// TIA Portal project "Project400 pid control implementation" (V20)

(* hardware
DEVICE "HMI_1"  KTP400 Basic PN
   slot 0: "HMI_1"  KTP400 Basic PN  6AV2 123-2DB03-0AX0  17.0.0.0
   slot 1: "HMI_RT_1"  KTP400 Basic PN  6AV2 123-2DB03-0AX0  17.0.0.0
   slot 5: "HMI_1.IE_CP_1"  PROFINET Interface  17.0.0.0
      slot 1: "PROFINET Interface_1"  PROFINET Interface
         slot 1: "Port_1"  Port
DEVICE "S7-1200 station_1"  S7-1200 Station
   slot 0: "Rack_0"  S7-1200 Rack  Rack  V1.0
   slot 1: "PLC_1"  CPU 1215C AC/DC/Rly  6ES7 215-1BG31-0XB0  V3.0
*)

// ===== PLC "PLC_1"  CPU 1215C AC/DC/Rly =====

VAR_GLOBAL   // PLC tag table "Default tag table"
   "Temperature_SP" AT %MD0 : Real;
   "Temperature_RV" AT %MD4 : Real;
   "Manual_output" AT %MD8 : Real;
   "Manual_mode" AT %M12.0 : Bool;
   "Scale_output" AT %MW14 : Word;
   "PID_on" AT %Q0.0 : Bool;
   "Man_pb" AT %M12.1 : Bool;
   "auto_pb" AT %M12.2 : Bool;
END_VAR

ORGANIZATION_BLOCK "Main"   // OB1, LAD, ProgramCycle
TITLE = "Main Program Sweep (Cycle)"
{ S7_Optimized_Access := 'TRUE' }
VERSION : 0.1
BEGIN

REGION Network 1: Auto/manual Controller
END_REGION

REGION Network 3
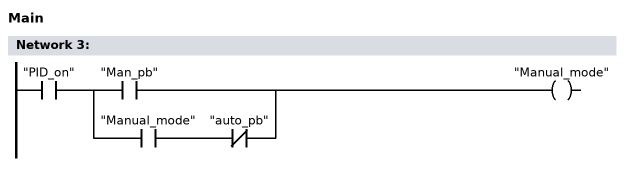
   RUNG wire#powerrail
      Contact( "PID_on" )
      wire#w1
      Contact( "Man_pb" )
      wire#w2
      Coil( "Manual_mode" )
   END_RUNG
   RUNG wire#w1
      Contact( "Manual_mode" )
      I_Contact( "auto_pb" )
   END_RUNG wire#w2
   // the same network as SCL:
   "Manual_mode" := "PID_on" AND ("Man_pb" OR ("Manual_mode" AND NOT "auto_pb"));
END_REGION
END_ORGANIZATION_BLOCK

ORGANIZATION_BLOCK "PID_CONTROLLER"   // OB30, LAD, CyclicInterrupt
{ S7_Optimized_Access := 'TRUE' }
VERSION : 0.1
BEGIN

REGION Network 1
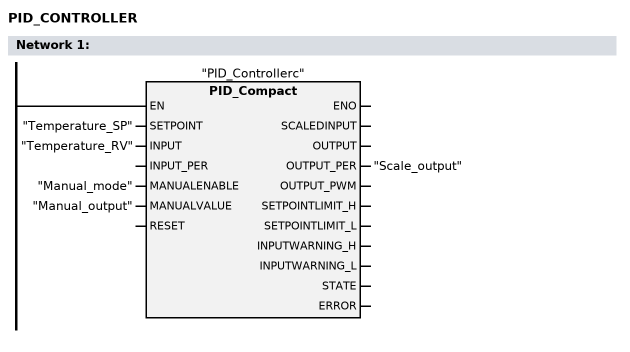
   "PID_Controllerc"(Setpoint := "Temperature_SP",   // PID_Compact
                     Input := "Temperature_RV",
                     ManualEnable := "Manual_mode",
                     ManualValue := "Manual_output",
                     Output_PER => "Scale_output");
END_REGION
END_ORGANIZATION_BLOCK

(* ===== HMI "HMI_RT_1" =====
system functions are stored by id; their names below are inferred from use
connection "HMI_Connection_1": ETHERNET, SMART_S7_1200_OMS

HMI tags "Default tag table"
   "Tag_ScreenNumber" : UInt, internal
   "Scale_output" : Word = PLC Scale_output AT %MW14, 1 s
   "Manual_output" : Real = PLC Manual_output AT %MD8, 1 s
   "Temperature_SP" : Real = PLC Temperature_SP AT %MD0, 1 s
   "Temperature_RV" : Real = PLC Temperature_RV AT %MD4, 1 s
   "auto_pb" : Bool = PLC auto_pb AT %M12.2, 1 s
   "Man_pb" : Bool = PLC Man_pb AT %M12.1, 1 s

Template "Template_1" 480x272
   Button "Exit" at 388,227 size 63x44; TextOff 'Exit'; PictureOff "ExitRuntime_KTP400_Basic_PN_TR"; PictureOn "ExitRuntime_KTP400_Basic_PN_TR"
      on Release: StopRuntime(0)
   Button "Template_Button" at 268,227 size 63x44; TextOff 'Text'
   Button "Template_Button_1" at 148,227 size 63x44; TextOff 'Text'
   Button "Start screen" at 28,227 size 63x44; TextOff 'Start screen'; PictureOff "NavigateHome_KTP400_Basic_PN_TR"; PictureOn "NavigateHome_KTP400_Basic_PN_TR"
      on Release: ActivateScreen("Root screen", 0)
   SymbolicIOField "Symbolic_IO_Field_Screen" at 82,8 size 311x29; TextOff '0'; TextOn '1'; TextList "TextList_ScreenNames"
      ProcessValue <- "Tag_ScreenNumber"
      on Change: ActivateScreenByNumber("Tag_ScreenNumber", 0)
   DateTimeField "HmiScreenItemData" at 395,22 size 85x22
   DateTimeField "HmiScreenItemData_1" at 395,0 size 85x22
   GraphicView "Logo" at 0,0 size 80x45; Picture "Logo of HMI_1"

screen "Root screen" 480x272, template "Template_1"
   on GenerateScreen: SetTag("Tag_ScreenNumber", 1)
   Bar "Bar_1" at 8,62 size 53x136; MinimumValue 0; MaximumValue 100
      ProcessValue <- "Scale_output"
   Bar "Bar_2" at 66,64 size 54x136; MinimumValue 0; MaximumValue 100
      ProcessValue <- "Manual_output"
   TextField "Text field_1" at 126,59 size 89x20; Text 'Temperature'
   TextField "Text field_2" at 131,99 size 102x20; Text 'Set Point Temp'
   SymbolicIOField "Symbolic I/O field_1" at 238,57 size 74x25; TextOff '0'; TextOn '1'
      ProcessValue <- "Temperature_RV"
   SymbolicIOField "Symbolic I/O field_2" at 237,109 size 73x27; TextOff '0'; TextOn '1'
      ProcessValue <- "Temperature_SP"
   SymbolicIOField "Symbolic I/O field_3" at 240,145 size 70x28; TextOff '0'; TextOn '1'
      ProcessValue <- "Scale_output"
   TextField "Text field_3" at 131,141 size 76x20; Text 'PID Output'
   SymbolicIOField "Symbolic I/O field_4" at 240,182 size 70x31; TextOff '0'; TextOn '1'
      ProcessValue <- "Manual_output"
   TextField "Text field_4" at 123,181 size 100x20; Text 'Manual Output'
   Button "Button_1" at 13,214 size 66x22; TextOff 'Auto'
      on Press: function_b14e0dd5("auto_pb", 0)
   Button "Button_2" at 96,212 size 66x22; TextOff 'Manual'
      on Press: function_b14e0dd5("Man_pb", 0)
   TextField "Text field_5" at 356,57 size 32x20; Text 'Gain'
   TextField "Text field_6" at 342,81 size 57x20; Text 'Integral'
   SymbolicIOField "Symbolic I/O field_5" at 405,53 size 74x25; TextOff '0'; TextOn '1'
      ProcessValue <- "Temperature_RV"
   SymbolicIOField "Symbolic I/O field_6" at 403,82 size 73x27; TextOff '0'; TextOn '1'
      ProcessValue <- "Temperature_SP"
   SymbolicIOField "Symbolic I/O field_7" at 403,117 size 70x28; TextOff '0'; TextOn '1'
      ProcessValue <- "Scale_output"
   TextField "Text field_7" at 328,116 size 72x20; Text 'Derivative'
*)